FUNCTION_BLOCK XABS_VIEW (* Abstract Superclass for a Transfer Component *)
  (* Standard: 61499-1 *)
  (* Version 0.1, 2004-09-01, JHC, Rockwell Automation, Changed DIA initial value to 0. *)
  (* Version 0.0, 2001-04-15, JHC, Rockwell Automation, Initial XML version. *)
  (* Compiler header: package fb.rt.hmi; *)
  (* Compiler Java IBM VisualAge 3.0 *)
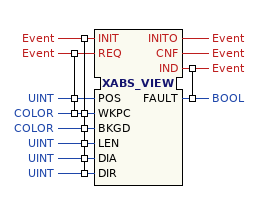
  EVENT_INPUT
    INIT WITH WKPC, BKGD, LEN, DIA, DIR; (* Initialize *)
    REQ WITH POS, WKPC; (* Update the display *)
  END_EVENT
  EVENT_OUTPUT
    INITO; (* Initialized *)
    CNF; (* Displayed *)
    IND WITH FAULT; (* Change in FAULT status *)
  END_EVENT
  VAR_INPUT
    POS : UINT; (* Position:0=HOME,100=END *)
    WKPC : COLOR := cyan; (* Workpiece Color *)
    BKGD : COLOR := blue; (* Transfer Bar Color *)
    LEN : UINT := 3; (* Bar Length in Diameters *)
    DIA : UINT; (* Workpiece diameter *)
    DIR : UINT; (* Orientation:0=L/R,1=T/B,2=R/L,3=B/T *)
  END_VAR
  VAR_OUTPUT
    FAULT : BOOL; (* 0=Normal,1=Fault *)
  END_VAR
  SERVICE XABS_VIEW/resource
    SEQUENCE init_new (* View component doesn't exist yet *)
      XABS_VIEW.INIT() -> resource.getNewView() -> resource.initView() -> XABS_VIEW.INITO();
    END_SEQUENCE
    SEQUENCE init_old (* View component exists *)
      XABS_VIEW.INIT() -> resource.initView() -> XABS_VIEW.INITO();
    END_SEQUENCE
    SEQUENCE normal_operation
      XABS_VIEW.REQ() -> resource.req() -> XABS_VIEW.CNF();
    END_SEQUENCE
    SEQUENCE fault_state_change
      resource.toggleFault() -> XABS_VIEW.IND();
    END_SEQUENCE
  END_SERVICE
END_FUNCTION_BLOCK
